TYPE ST_TableBottlePlace :
STRUCT
	sProductName:STRING;
	nBottleType:nBottleTypes;
	nState: nTableBottlePlaceState;
	byDetectionStatus: BYTE;
	iCurrentPosition: USINT;
	iPlaceNumber: USINT;
END_STRUCT
END_TYPE

(* stored: Version 1.1.0.1, ProductVersion 3.1.4024.15
   DUT ST_TableBottlePlace: Id {59226ff1-7df5-43ed-98cb-c70a30f0ca6e} *)
